// TIA Portal V15.1 export
// export: Created 2024-06-21T08:41:11.4906908Z, ExportSetting WithDefaults, DisplayName Totally Integrated Automation Portal, DisplayVersion V15.1 Update 5, DisplayName TIA Portal Openness, DisplayVersion V15.1 Update 5, DisplayName SINAMICS Startdrive Advanced, DisplayVersion V15.1, DisplayName G130, G150, S120, S150, SINAMICS MV, S210, DisplayVersion V15.1, DisplayName G110M, G120, G120C, G120D, G120P, DisplayVersion V15.1, DisplayName STEP 7 Professional, DisplayVersion V15.1 Update 5, DisplayName STEP 7 Safety, DisplayVersion V15.1, DisplayName WinCC Professional, DisplayVersion V15.1 Update 5, DisplayName SIMATIC Visualization Architect, DisplayVersion V15.1
FUNCTION "LGBBuhlLock-Config" : Void   // FC6630, FBD
TITLE = LMovUnit2Pos1S-C-Config / LGBBuhlLock-Config
{ S7_Optimized_Access := 'FALSE' }
AUTHOR : VCC
FAMILY : Control
NAME : Bit2Word
VERSION : 1.0
// =============================================================================
// Move Configuration 
// =============================================================================
// stored: AutoNumber false, IsIECCheckEnabled false, SetENOAutomatically False, UDAEnableTagReadback false
   VAR_INPUT
      C_AlarmResetUsed : Bool;   // Set position / If true, the Alarms will be stored untill reseted
      C_EnableMemBegin : Bool;   // Reset position / Enable memory Begin (Command Request is memorised until pos reached)
      C_EnIntlkAlm : Bool;   // Active / Enable interlock Alarm
      C_KeepPosition : Bool;   // Invisible / If true, the last position shall be kept ON and checked
      C_EnableAlarm : Bool;   // Object out of use / Enable Alarm
      C_EnAlmOvertime : Bool;   // Object out of use / Enable Alarm
      C_AlarmHighSeverity : Bool;   // Interlock alarm for Set direction / Alarm severity
      C_SafetySwUsed : Bool;   // Safety switch used
      C_SafetySwNc : Bool;   // Safety switch NC contact
      C_MotorProtectionUsed : Bool;   // Motor Protection used
      C_MotorProtectionNc : Bool;   // Motor Protection NC contact
      C_SetReset : Bool;   // Set Reset
      C_ManualClampCmdSet : Bool;   // Manual Clamp Command Set
      C_ManualClampCmdReset : Bool;   // Manual Clamp Command Reset
      C_ForceManual : Bool;   // Force Manual
      C_RunTimeMaxSetWarn : DInt;   // Maximum Time (x1ms) that the function may run (create overtime) / Maximum Time (x1ms) that the function may run (create Overtime)
      C_RunTimeMaxSetAlarm : DInt;   // Maximum Time (x1ms) that the function may run (create overtime) / Maximum Time (x1ms) that the function may run (create Overtime)
      C_RunTimeMaxResWarn : DInt;   // Maximum Time (x1ms) that the function may run (create overtime) / Maximum Time (x1ms) that the function may run (create Overtime)
      C_RunTimeMaxResAlarm : DInt;   // Maximum Time (x1ms) that the function may run (create overtime) / Maximum Time (x1ms) that the function may run (create Overtime)
      C_TimeAlmFilt : DInt;   // Timer before any actuator alarm will be active (welding..) / Timer before any actuator Alarm will be active (welding..)
   END_VAR
   VAR_IN_OUT
      IO_Config : "MovConfig";   // Output Word / Config
   END_VAR
BEGIN

REGION Network 1: **** 1 - Inputs **** Configuration
   // Configuration
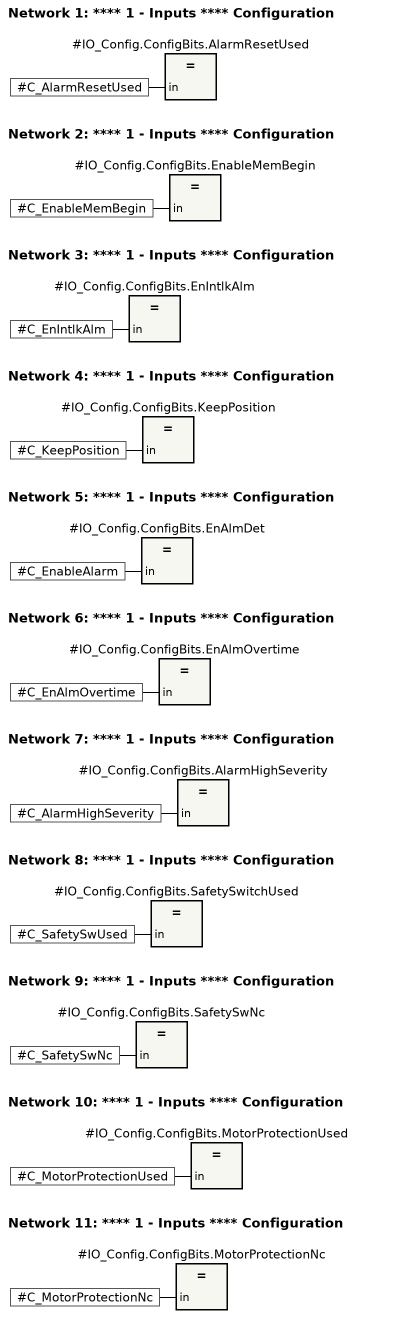
   #IO_Config.ConfigBits.AlarmResetUsed := #C_AlarmResetUsed;
END_REGION

REGION Network 2: **** 1 - Inputs **** Configuration
   // Configuration
   #IO_Config.ConfigBits.EnableMemBegin := #C_EnableMemBegin;
END_REGION

REGION Network 3: **** 1 - Inputs **** Configuration
   // Configuration
   #IO_Config.ConfigBits.EnIntlkAlm := #C_EnIntlkAlm;
END_REGION

REGION Network 4: **** 1 - Inputs **** Configuration
   // Configuration
   #IO_Config.ConfigBits.KeepPosition := #C_KeepPosition;
END_REGION

REGION Network 5: **** 1 - Inputs **** Configuration
   // Configuration
   #IO_Config.ConfigBits.EnAlmDet := #C_EnableAlarm;
END_REGION

REGION Network 6: **** 1 - Inputs **** Configuration
   // Configuration
   #IO_Config.ConfigBits.EnAlmOvertime := #C_EnAlmOvertime;
END_REGION

REGION Network 7: **** 1 - Inputs **** Configuration
   // Configuration
   #IO_Config.ConfigBits.AlarmHighSeverity := #C_AlarmHighSeverity;
END_REGION

REGION Network 8: **** 1 - Inputs **** Configuration
   // Configuration
   #IO_Config.ConfigBits.SafetySwitchUsed := #C_SafetySwUsed;
END_REGION

REGION Network 9: **** 1 - Inputs **** Configuration
   // Configuration
   #IO_Config.ConfigBits.SafetySwNc := #C_SafetySwNc;
END_REGION

REGION Network 10: **** 1 - Inputs **** Configuration
   // Configuration
   #IO_Config.ConfigBits.MotorProtectionUsed := #C_MotorProtectionUsed;
END_REGION

REGION Network 11: **** 1 - Inputs **** Configuration
   // Configuration
   #IO_Config.ConfigBits.MotorProtectionNc := #C_MotorProtectionNc;
END_REGION

REGION Network 12: **** 1 - Inputs **** Configuration
   // Move bit 15Configuration
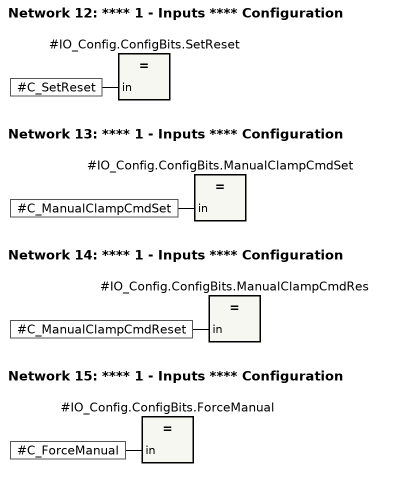
   #IO_Config.ConfigBits.SetReset := #C_SetReset;
END_REGION

REGION Network 13: **** 1 - Inputs **** Configuration
   // Configuration
   #IO_Config.ConfigBits.ManualClampCmdSet := #C_ManualClampCmdSet;
END_REGION

REGION Network 14: **** 1 - Inputs **** Configuration
   // Configuration
   #IO_Config.ConfigBits.ManualClampCmdRes := #C_ManualClampCmdReset;
END_REGION

REGION Network 15: **** 1 - Inputs **** Configuration
   // Configuration
   #IO_Config.ConfigBits.ForceManual := #C_ForceManual;
END_REGION

NETWORK
TITLE = **** 1 Inputs **** Move Config UDT
// Move Config
      L     #C_RunTimeMaxSetWarn;
      T     #IO_Config.RunTimeMaxSetWarn;
      L     #C_RunTimeMaxSetAlarm;
      T     #IO_Config.RunTimeMaxSetAlm;
      L     #C_RunTimeMaxResWarn;
      T     #IO_Config.RunTimeMaxResWarn;
      L     #C_RunTimeMaxResAlarm;
      T     #IO_Config.RunTimeMaxResAlm;
      L     #C_TimeAlmFilt;
      T     #IO_Config.TimeAlmFilt;
END_FUNCTION
